Staubli VAL3: _recordLoc.pgx

program _recordLoc(tool x_tool (dimensions=1), frame x_frame (dimensions=1), trsf& x_TRSF[] (dimensions=1), config& x_CFG[] (dimensions=1))
begin
  // This program records the position and the configuration
  // of the robot's tool in the frame passed as parameter.
  //
  // Input Param
  //  x_frame : reference frame in which position must be recorded
  //  x_tool  :
  //
  // Output Param
  // x_TRSF : Position
  // x_CFG  : Configuration
  //
  // Created 16-01-06                                   C.CURRIVAND
  //----------------------------------------------------------------
  x_TRSF=position(here(x_tool,x_frame),x_frame)
  x_CFG=config(herej())
end
